{attribute 'qualified_only'}
{attribute 'strict'}
TYPE E_RotationDirection :
(
	NONE,
	EDGE_DETECTED
);
END_TYPE

(* stored: Version 1.1.0.1, ProductVersion 3.1.4024.11
   DUT E_RotationDirection: Id {6a71a329-4637-4add-bee6-0259faed9aad} *)
